"A_2760_MXZ02_O1"	Q 765.7	BOOL	// GERM FAN 2
"A_2801_MXZ01_O1"	Q 802.0	BOOL	// BELT CONVEYOR
"A_2802_MXZ01_O1"	Q 802.1	BOOL	// CHUTE DRIVE LEFT SIDE
"A_2802_MXZ01_O2"	Q 802.2	BOOL	// CHUTE DRIVE RIGHT SIDE
"A_2811_MXZ61_O1"	Q 803.2	BOOL	// TURNING SCREW DRIVE 1
"A_2811_MXZ62_O1"	Q 803.3	BOOL	// TURNING SCREW DRIVE 2
"A_2811_MXZ63_O1"	Q 803.4	BOOL	// TURNING SCREW DRIVE 3
"A_2811_MXZ64_O1"	Q 803.5	BOOL	// TURNING SCREW DRIVE 4
"A_2811_MXZ65_O1"	Q 803.6	BOOL	// TURNING SCREW DRIVE 5
"A_2811_MXZ66_O1"	Q 803.7	BOOL	// TURNING SCREW DRIVE 6
"A_2811_MXZ67_O1"	Q 804.0	BOOL	// TURNING SCREW DRIVE 7
"A_2811_MXZ68_O1"	Q 804.1	BOOL	// TURNING SCREW DRIVE 8
"A_2811_MXZ69_O1"	Q 804.2	BOOL	// TURNING SCREW DRIVE 9
"A_2811_MXZ70_O1"	Q 804.3	BOOL	// TURNING SCREW DRIVE 10
"A_2811_MXZ71_O1"	Q 804.4	BOOL	// TURNING SCREW DRIVE 11
"A_2811_MXZ72_O1"	Q 804.5	BOOL	// TURNING SCREW DRIVE 12
"A_2811_MXZ73_O1"	Q 804.6	BOOL	// TURNING SCREW DRIVE 13
"A_2815_MXZ11_O1"	Q 808.0	BOOL	// HORIZONTAL SCREW
"A_2815_MXZ15_O1"	Q 808.2	BOOL	// LIFTING SCREW
"A_2815_MXZ21_O1"	Q 808.3	BOOL	// LIFTING DEVICE DOWN
"A_2815_MXZ21_O2"	Q 808.4	BOOL	// LIFTING DEVICE UP
"A_2845_QXV21_O1"	Q 816.0	BOOL	// START COOLING UNIT GERMINATING
"A_2845_QXV31_O1"	Q 816.1	BOOL	// START COOLING UNIT GERMINATING
"A_2801_QXV21_O1"	Q 816.2	BOOL	// BALL VALVE SPRAY WATER OPEN
"A_2816_QXV12_O2"	Q 816.4	BOOL	// BALL VALVE SPRINKING WATER LINE
"A_2831_QXV12_O1"	Q 816.6	BOOL	// BALL VALVE AIR HUMIDIFICATION
"A_2831_QXV22_O1"	Q 816.7	BOOL	// BALL VALVE AIR HUMIDIFICATION
"A_2831_QXV12_O2"	Q 817.2	BOOL	// BALL VALVE VALVE HUMIDIFICATION
"A_2899_PAZ11_O1"	Q 818.0	BOOL	// ALARM HORN MACHINE
"A_2812_QXV12_O2"	Q 840.0	BOOL	// BALL VALVE SPRINKING WATER LINE 1
"A_28_A408Z1_O1"	Q 840.1	BOOL	// RESET ALARM
"A_2811_KCL01_O1"	Q 840.4	BOOL	// ALARM FLASHER
"A_2811_KCL01_O2"	Q 840.5	BOOL	// SPARE
"A_2811_MXZ21_O1"	Q 841.0	BOOL	// COUPLING DRIVE
"A_2811_MXZ21_O2"	Q 841.1	BOOL	// COUPLING DRIVE
"A_2811_MXZ25_O1"	Q 841.2	BOOL	// COUPLING DRIVE
"A_2811_MXZ25_O2"	Q 841.3	BOOL	// COUPLING DRIVE
"A_2811_MXZ31_O1"	Q 841.4	BOOL	// COUPLING DRIVE
"A_2811_MXZ31_O2"	Q 841.5	BOOL	// COUPLING DRIVE
"A_2811_MXZ35_O1"	Q 841.6	BOOL	// COUPLING DRIVE
"A_2811_MXZ35_O2"	Q 841.7	BOOL	// COUPLING DRIVE
"A_2815_KCL01_O1"	Q 860.0	BOOL	// BACKWALL LIFTED
"A_2815_KCL01_O2"	Q 860.1	BOOL	// BACKWALL LOWERED
"A_2815_KCL01_O3"	Q 860.2	BOOL	// UNCOUPLED
"A_2815_KCL01_O4"	Q 860.3	BOOL	// COUPLED
"A_2815_KCL01_O5"	Q 860.4	BOOL	// WALL LOCKED
"A_2815_KCL01_O6"	Q 860.5	BOOL	// WALL UNLOCKED
"A_2815_KCL01_O7"	Q 860.6	BOOL	// CLEANING FLAP 1/2
"A_2815_MXZ41_O1"	Q 861.0	BOOL	// COUPLING DRIVE
"A_2815_MXZ41_O2"	Q 861.1	BOOL	// COUPLING DRIVE
"A_2815_MXZ45_O1"	Q 861.2	BOOL	// COUPLING DRIVE
"A_2815_MXZ45_O2"	Q 861.3	BOOL	// COUPLING DRIVE
"A_2850_MXZ01_O1"	Q 864.0	BOOL	// AIR-FLAP 1 OPEN
"A_2850_MXZ01_O2"	Q 864.1	BOOL	// AIR-FLAP 1 CLOSE
"A_2851_MXZ01_O1"	Q 864.4	BOOL	// AIR-FLAP 2 OPEN
"A_2851_MXZ01_O2"	Q 864.5	BOOL	// AIR-FLAP 2 CLOSE
"A_2852_MXZ01_O1"	Q 865.0	BOOL	// AIR-FLAP 3 OPEN
"A_2852_MXZ01_O2"	Q 865.1	BOOL	// AIR-FLAP 3 CLOSE
"A_2854_MXZ01_O1"	Q 865.4	BOOL	// WATER PUMP 1
"A_2855_MXZ01_O1"	Q 865.5	BOOL	// WATER PUMP 2
"A_2860_MXZ01_O1"	Q 865.6	BOOL	// GERM FAN 1
"A_2860_MXZ02_O1"	Q 865.7	BOOL	// GERM FAN 2
"A_3111_MXZ11_O1"	Q 900.0	BOOL	// UN-/LOADING SCREW DISCHARGE
"A_3111_MXZ21_O1"	Q 900.1	BOOL	// LIFTING DRIVE 1 INSIDE LOWERING
"A_3111_MXZ21_O2"	Q 900.2	BOOL	// LIFTING DRIVE 1 INSIDE LIFTING
"A_3111_MXZ31_O1"	Q 900.3	BOOL	// LIFTING DRIVE 2 OUTSIDE LOWERING
"A_3111_MXZ31_O2"	Q 900.4	BOOL	// LIFTING DRIVE 2 OUTSIDE LIFTING
"A_3111_MXZ41_O1"	Q 900.5	BOOL	// TRAVELING DRIVE
"A_3115_MXZ11_O1"	Q 900.6	BOOL	// DISCHARGE FLAP CLOSE
"A_3115_MXZ11_O2"	Q 900.7	BOOL	// DISCHARGE FLAP OPEN
"A_3135_MXZ11_O1"	Q 901.0	BOOL	// LOUVER RECYCLE AIR 1 CLOSE
"A_3135_MXZ11_O2"	Q 901.1	BOOL	// LOUVER RECYCLE AIR 1 OPEN
"A_3136_MXZ11_O1"	Q 901.2	BOOL	// LOUVER RECYCLE AIR 2 CLOSE
"A_3136_MXZ11_O2"	Q 901.3	BOOL	// LOUVER RECYCLE AIR 2 OPEN
"A_3140_MXZ11_O1"	Q 901.4	BOOL	// LOUVER RECYCLE AIR 1 CLOSE
"A_3140_MXZ11_O2"	Q 901.5	BOOL	// LOUVER RECYCLE AIR 1 OPEN
"A_3141_MXZ11_O1"	Q 901.6	BOOL	// LOUVER RECYCLE AIR 2 CLOSE
"A_3141_MXZ11_O2"	Q 901.7	BOOL	// LOUVER RECYCLE AIR 2 OPEN
"A_3145_MXZ11_O1"	Q 902.0	BOOL	// LOUVER WITHERING AIR 1 CLOSE
"A_3145_MXZ11_O2"	Q 902.1	BOOL	// LOUVER WITHERING AIR 1 OPEN
"A_3146_MXZ11_O1"	Q 902.2	BOOL	// LOUVER WITHERING AIR 2 CLOSE
"A_3146_MXZ11_O2"	Q 902.3	BOOL	// LOUVER WITHERING AIR 2 OPEN
"A_3150_MXZ11_O1"	Q 902.4	BOOL	// LOUVER FRESH AIR 1 CLOSE
"A_3150_MXZ11_O2"	Q 902.5	BOOL	// LOUVER FRESH AIR 1 OPEN
"A_3151_MXZ11_O1"	Q 902.6	BOOL	// LOUVER FRESH AIR 2 CLOSE
"A_3151_MXZ11_O2"	Q 902.7	BOOL	// LOUVER FRESH AIR 2 OPEN
"A_3152_MXZ11_O1"	Q 903.0	BOOL	// LOUVER FRESH AIR 3 CLOSE
"A_3152_MXZ11_O2"	Q 903.1	BOOL	// LOUVER FRESH AIR 3 OPEN
"A_3153_MXZ11_O1"	Q 903.2	BOOL	// LOUVER FRESH AIR 4 CLOSE
"A_3153_MXZ11_O2"	Q 903.3	BOOL	// LOUVER FRESH AIR 4 OPEN
"A_3158_MXZ11_O1"	Q 903.4	BOOL	// LOUVER AIR HEATER 1 CLOSE
"A_3158_MXZ11_O2"	Q 903.5	BOOL	// LOUVER AIR HEATER 1 OPEN
"A_3159_MXZ11_O1"	Q 903.6	BOOL	// LOUVER AIR HEATER 2 CLOSE
"A_3159_MXZ11_O2"	Q 903.7	BOOL	// LOUVER AIR HEATER 2 OPEN
"A_3101_MXZ01_O1"	Q 904.0	BOOL	// OUTLET FLAP DRIVE CLOSE
"A_3101_MXZ01_O2"	Q 904.1	BOOL	// OUTLET FLAP DRIVE OPEN
"A_3161_KCL11_O1"	Q 916.0	BOOL	// BURNER 1 MAIN FAN RUNNING
"A_3161_KCL11_O2"	Q 916.1	BOOL	// BURNER 1 EXTERAL ON
"A_3161_KCL12_O1"	Q 917.0	BOOL	// BURNER 2 MAIN FAN RUNNING
"A_3161_KCL12_O2"	Q 917.1	BOOL	// BURNER 2 EXTERAL ON
"A_3199_PAZ11_O1"	Q 924.0	BOOL	// ALARM HORN
"A_3211_MXZ11_O1"	Q 1000.0	BOOL	// UN-/LOADING SCREW DISCHARGE
"A_3211_MXZ21_O1"	Q 1000.1	BOOL	// LIFTING DRIVE 1 INSIDE LOWERING
"A_3211_MXZ21_O2"	Q 1000.2	BOOL	// LIFTING DRIVE 1 INSIDE LIFTING
"A_3211_MXZ31_O1"	Q 1000.3	BOOL	// LIFTING DRIVE 2 OUTSIDE LOWERING
"A_3211_MXZ31_O2"	Q 1000.4	BOOL	// LIFTING DRIVE 2 OUTSIDE LIFTING
"A_3211_MXZ41_O1"	Q 1000.5	BOOL	// TRAVELING DRIVE
"A_3215_MXZ11_O1"	Q 1000.6	BOOL	// DISCHARGE FLAP CLOSE
"A_3215_MXZ11_O2"	Q 1000.7	BOOL	// DISCHARGE FLAP OPEN
"A_3235_MXZ11_O1"	Q 1001.0	BOOL	// LOUVER RECYCLE AIR 1 CLOSE
"A_3235_MXZ11_O2"	Q 1001.1	BOOL	// LOUVER RECYCLE AIR 1 OPEN
"A_3236_MXZ11_O1"	Q 1001.2	BOOL	// LOUVER RECYCLE AIR 2 CLOSE
"A_3236_MXZ11_O2"	Q 1001.3	BOOL	// LOUVER RECYCLE AIR 2 OPEN
"A_3240_MXZ11_O1"	Q 1001.4	BOOL	// LOUVER RECYCLE AIR 1 CLOSE
"A_3240_MXZ11_O2"	Q 1001.5	BOOL	// LOUVER RECYCLE AIR 1 OPEN
"A_3241_MXZ11_O1"	Q 1001.6	BOOL	// LOUVER RECYCLE AIR 2 CLOSE
"A_3241_MXZ11_O2"	Q 1001.7	BOOL	// LOUVER RECYCLE AIR 2 OPEN
"A_3245_MXZ11_O1"	Q 1002.0	BOOL	// LOUVER WITHERING AIR 1 CLOSE
"A_3245_MXZ11_O2"	Q 1002.1	BOOL	// LOUVER WITHERING AIR 1 OPEN
"A_3246_MXZ11_O1"	Q 1002.2	BOOL	// LOUVER WITHERING AIR 2 CLOSE
"A_3246_MXZ11_O2"	Q 1002.3	BOOL	// LOUVER WITHERING AIR 2 OPEN
"A_3250_MXZ11_O1"	Q 1002.4	BOOL	// LOUVER FRESH AIR 1 CLOSE
"A_3250_MXZ11_O2"	Q 1002.5	BOOL	// LOUVER FRESH AIR 1 OPEN
"A_3251_MXZ11_O1"	Q 1002.6	BOOL	// LOUVER FRESH AIR 2 CLOSE
"A_3251_MXZ11_O2"	Q 1002.7	BOOL	// LOUVER FRESH AIR 2 OPEN
"A_3252_MXZ11_O1"	Q 1003.0	BOOL	// LOUVER FRESH AIR 3 CLOSE
"A_3252_MXZ11_O2"	Q 1003.1	BOOL	// LOUVER FRESH AIR 3 OPEN
"A_3253_MXZ11_O1"	Q 1003.2	BOOL	// LOUVER FRESH AIR 4 CLOSE
"A_3253_MXZ11_O2"	Q 1003.3	BOOL	// LOUVER FRESH AIR 4 OPEN
"A_3258_MXZ11_O1"	Q 1003.4	BOOL	// LOUVER AIR HEATER 1 CLOSE
"A_3258_MXZ11_O2"	Q 1003.5	BOOL	// LOUVER AIR HEATER 1 OPEN
"A_3259_MXZ11_O1"	Q 1003.6	BOOL	// LOUVER AIR HEATER 2 CLOSE
"A_3259_MXZ11_O2"	Q 1003.7	BOOL	// LOUVER AIR HEATER 2 OPEN
"A_3201_MXZ01_O1"	Q 1004.0	BOOL	// OUTLET FLAP DRIVE CLOSE
"A_3201_MXZ01_O2"	Q 1004.1	BOOL	// OUTLET FLAP DRIVE OPEN
"A_3261_KCL11_O1"	Q 1016.0	BOOL	// BURNER 3 MAIN FAN RUNNING
"A_3261_KCL11_O2"	Q 1016.1	BOOL	// BURNER 3 EXTERAL ON
"A_3299_PAZ11_O1"	Q 1024.0	BOOL	// ALARM HORN
"A_1911_MXZ01_O1"	Q 1102.0	BOOL	// BELT CONVEYOR
"A_1915_MXZ01_O1"	Q 1102.1	BOOL	// BELT CONVEYOR
"A_1921_MXZ01_O1"	Q 1102.2	BOOL	// BELT CONVEYOR
"A_1931_MXZ01_O1"	Q 1102.3	BOOL	// BELT CONVEYOR
"A_1941_MXZ01_O1"	Q 1102.4	BOOL	// BELT CONVEYOR
"A_1942_MXZ01_O3"	Q 1102.5	BOOL	// CHUTE DRIVE LOW ROTARY SPEED
"A_1942_MXZ01_O1"	Q 1102.6	BOOL	// CHUTE DRIVE LEFT SIDE
"A_1942_MXZ01_O2"	Q 1102.7	BOOL	// CHUTE DRIVE RIGHT SIDE
"A_1999_PAZ11_O1"	Q 1104.0	BOOL	// ALARM HORN
"A_1911_QXV31_O1"	Q 1108.0	BOOL	// BALL VALVE SPRAY WATER OPEN
"A_1915_QXV31_O1"	Q 1108.1	BOOL	// BALL VALVE SPRAY WATER OPEN
"A_1921_QXV31_O1"	Q 1108.2	BOOL	// BALL VALVE SPRAY WATER OPEN
"A_2911_MXZ01_O1"	Q 1118.0	BOOL	// BELT CONVEYOR
"A_2914_MXZ01_O1"	Q 1118.1	BOOL	// BELT CONVEYOR
"A_2917_MXZ01_O1"	Q 1118.2	BOOL	// BELT CONVEYOR
"A_2920_MXZ01_O1"	Q 1118.3	BOOL	// BELT CONVEYOR
"A_2923_MXZ01_O1"	Q 1118.4	BOOL	// BELT CONVEYOR
"A_2926_MXZ01_O1"	Q 1118.5	BOOL	// BELT CONVEYOR
"A_2929_MXZ01_O1"	Q 1118.6	BOOL	// BELT CONVEYOR
"A_2932_MXZ01_02_O1"	Q 1119.1	BOOL	// BELT CONVEYOR DRIVE 1/2
"A_2935_MXZ01_O1"	Q 1119.2	BOOL	// BELT CONVEYOR RIGHT
"A_2935_MXZ01_O2"	Q 1119.3	BOOL	// BELT CONVEYOR LEFT
"A_2999_PAZ11_O1"	Q 1120.0	BOOL	// ALARM HORN
"A_2911_QXV31_O1"	Q 1124.0	BOOL	// BALL VALVE SPRAY WATER OPEN
"A_2914_QXV31_O1"	Q 1124.1	BOOL	// BALL VALVE SPRAY WATER OPEN
"A_2917_QXV31_O1"	Q 1124.2	BOOL	// BALL VALVE SPRAY WATER OPEN
"A_2920_QXV31_O1"	Q 1124.3	BOOL	// BALL VALVE SPRAY WATER OPEN
"A_2923_QXV31_O1"	Q 1124.4	BOOL	// BALL VALVE SPRAY WATER OPEN
"A_2935_QXV31_O1"	Q 1124.6	BOOL	// BALL VALVE SPRAY WATER OPEN
"A_2935_QXV41_O1"	Q 1124.7	BOOL	// BALL VALVE SPRAY WATER OPEN
"A_3911_MXZ01_O1"	Q 1134.0	BOOL	// CHAIN CONVEYOR
"A_3912_MXZ01_O1"	Q 1134.1	BOOL	// OUTLET FLAP DRIVE CLOSE
"A_3912_MXZ01_O2"	Q 1134.2	BOOL	// OUTLET FLAP DRIVE OPEN
"A_3914_MXZ01_O1"	Q 1134.3	BOOL	// FAN DRIVE "NOTUSED"
"A_3921_MXZ01_O1"	Q 1134.4	BOOL	// CHAIN CONVEYOR
"A_3922_MXZ01_O1"	Q 1134.5	BOOL	// OUTLET FLAP DRIVE CLOSE
"A_3922_MXZ01_O2"	Q 1134.6	BOOL	// OUTLET FLAP DRIVE OPEN
"A_3924_MXZ01_O1"	Q 1134.7	BOOL	// FAN DRIVE "NOTUSED"
"A_3930_MXZ01_O1"	Q 1135.0	BOOL	// ELEVATOR
"A_3932_MXZ01_O1"	Q 1135.1	BOOL	// FAN DRIVE "NOTUSED"
"A_3935_MXZ01_O1"	Q 1135.2	BOOL	// FLAP BOX DRIVE RIGHT SIDE
"A_3935_MXZ01_O2"	Q 1135.3	BOOL	// FLAP BOX DRIVE LEFT SIDE
"A_3938_MXZ01_O1"	Q 1135.4	BOOL	// BELT CONVEYOR
"A_3945_MXZ01_O1"	Q 1135.5	BOOL	// ELEVATOR
"A_3952_MXZ01_O1"	Q 1135.6	BOOL	// DISCHARGER DMBG DRIVE
"A_3955_MXZ01_O1"	Q 1135.7	BOOL	// SCREW CONVEYOR DRIVE
"A_3952_XCJ20_O1"	Q 1136.0	BOOL	// VALVE DMBG CLOSE
"A_3952_XCJ20_O2"	Q 1136.1	BOOL	// VALVE DMBG OPEN
"A_3952_XCJ20_O3"	Q 1136.2	BOOL	// VALVE DMBG CLOSE
"A_3952_XCJ20_O4"	Q 1136.3	BOOL	// VALVE DMBG OPEN
"A_3960_MXZ01_O1"	Q 1136.4	BOOL	// FAN DRIVE
"A_3965_MXZ01_O1"	Q 1136.5	BOOL	// AIRLOCK
"A_3970_MXZ01_O1"	Q 1136.6	BOOL	// AIRLOCK
"A_3999_PAZ11_O1"	Q 1137.0	BOOL	// ALARM HORN
"A_3913_KFC10_O1"	Q 1140.0	BOOL	// FILTER ASPIRATION ON "NOTUSED"
"A_3923_KFC10_O1"	Q 1140.1	BOOL	// FILTER ASPIRATION ON "NOTUSED"
"A_3931_KFC10_O1"	Q 1140.2	BOOL	// FILTER ASPIRATION ON "NOTUSED"
"A_3956_KCL01_O2"	Q 1140.4	BOOL	// LIGHT CUSTOMER ON
"A_3956_KCL01_O3"	Q 1140.5	BOOL	// LIGHT CUSTOMER OFF
"A_3956_KCL01_O1"	Q 1140.6	BOOL	// TURN ON EXCISTING DEGERMINATING SYSTEM
"A_2145_QXV21_AO1"	QW 168	WORD	// REGULATING VALVE SET POINT
"A_2145_QXV31_AO1"	QW 170	WORD	// REGULATING VALVE SET POINT
"A_2245_QXV21_AO1"	QW 268	WORD	// REGULATING VALVE SET POINT
"A_2245_QXV31_AO1"	QW 270	WORD	// REGULATING VALVE SET POINT
"A_2345_QXV21_AO1"	QW 368	WORD	// REGULATING VALVE SET POINT
"A_2345_QXV31_AO1"	QW 382	WORD	// REGULATING VALVE SET POINT
"A_2445_QXV21_AO1"	QW 468	WORD	// REGULATING VALVE SET POINT
"A_2445_QXV31_AO1"	QW 482	WORD	// REGULATING VALVE SET POINT
"CTUD"	SFB 2	SFB 2	// Count Up / Down
"TON"	SFB 4	SFB 4	// Generate an On Delay
"SIEMENS_BSEND"	SFB 12	SFB 12	// SIEMENS: Block Oriented Send
"SIEMENS_BRCV"	SFB 13	SFB 13	// SIEMENS: Block Oriented Receive
"SIEMENS_HS_COUNT"	SFB 29	SFB 29	// SIEMENS: High-Speed Counter (CPU 312, Integrated Function)
"SIEMENS_FREQ_MES"	SFB 30	SFB 30	// SIEMENS: Frequency Meter (CPU 312, Integrated Function)
"SIEMENS_POSITION"	SFB 31	SFB 31	// SIEMENS: Open-Loop Positioning (CPU 312, Integrated Function)
"SIEMENS_SET_CLK"	SFC 0	SFC 0	// SIEMENS: Set System Clock
"SIEMENS_READ_CLK"	SFC 1	SFC 1	// SIEMENS: Read System Clock
"SIEMENS_SET_RTM"	SFC 2	SFC 2	// SIEMENS: Set Run-Time Meter
"SIEMENS_CTRL_RTM"	SFC 3	SFC 3	// SIEMENS: Start/Stop Run-Time Meter
"SIEMENS_READ_RTM"	SFC 4	SFC 4	// SIEMENS: Read Run-Time Meter
"GADR_LGC"	SFC 5	SFC 5	// Query Logical Address of a Channel
"RD_SINFO"	SFC 6	SFC 6	// Read OB Start Information
"DPNRM_DG"	SFC 13	SFC 13	// Read Diagnostic Data of a DP Slave
"SIEMENS_DPRD_DAT"	SFC 14	SFC 14	// SIEMENS: Read data for DP-Node
"SIEMENS_DPWR_DAT"	SFC 15	SFC 15	// SIEMENS: Write Data to DP-Node
"SIEMENS_BLKMOV"	SFC 20	SFC 20	// SIEMENS: Direct Word Move
"SIEMENS_FILL"	SFC 21	SFC 21	// SIEMENS: Initialize a memory area
"SIEMENS_CREAT_DB"	SFC 22	SFC 22	// SIEMENS: Create Data Block
"SIEMENS_TEST_DB"	SFC 24	SFC 24	// SIEMENS: Test DB
"SIEMENS_SET_TINT"	SFC 28	SFC 28	// SIEMENS: Set Time-of-Day Interrupt
"SIEMENS_CAN_TINT"	SFC 29	SFC 29	// SIEMENS: Cancel Time-of-Day Interrupt
"SIEMENS_ACT_TINT"	SFC 30	SFC 30	// SIEMENS: Activate Time-of-Day Interrupt
"SIEMENS_QRY_TINT"	SFC 31	SFC 31	// SIEMENS: Query Time-of-Day Interrupt
"SIEMENS_SRT_DINT"	SFC 32	SFC 32	// SIEMENS: Start Time-Delay Interrupt
"SIEMENS_CAN_DINT"	SFC 33	SFC 33	// SIEMENS: Cancel Time-Delay Interrupt
"SIEMENS_QRY_DINT"	SFC 34	SFC 34	// SIEMENS: Query Time-Delay Interrupt
"SIEMENS_MSK_FLT"	SFC 36	SFC 36	// SIEMENS: Mask synchronous faults
"SIEMENS_DMSK_FLT"	SFC 37	SFC 37	// SIEMENS: Unmask Synchronous Faults
"SIEMENS_READ_ERR"	SFC 38	SFC 38	// SIEMENS: Read Error Registers
"SIEMENS_DIS_IRT"	SFC 39	SFC 39	// SIEMENS: Disable Interrupt
"SIEMENS_EN_IRT"	SFC 40	SFC 40	// SIEMENS: Enable New Interrupts and Asynchronous Errors
"SIEMENS_DIS_AIRT"	SFC 41	SFC 41	// SIEMENS: Disable Alarm Interrupts
"SIEMENS_EN_AIRT"	SFC 42	SFC 42	// SIEMENS: Enable Alarm Interrupts
"SIEMENS_RE_TRIGR"	SFC 43	SFC 43	// SIEMENS: Retrigger Cycle Time Monitoring
"SIEMENS_REPL_VAL"	SFC 44	SFC 44	// SIEMENS: Replace Value
"SIEMENS_STP"	SFC 46	SFC 46	// SIEMENS: Change the CPU to STOP
"SIEMENS_WAIT"	SFC 47	SFC 47	// SIEMENS: Wait
"SIEMENS_LGC_GADR"	SFC 49	SFC 49	// SIEMENS:
"SIEMENS_RD_LGADR"	SFC 50	SFC 50	// SIEMENS:
"SIEMENS_RDSYSST"	SFC 51	SFC 51	// SIEMENS: Read System Status
"SIEMENS_WR_USMSG"	SFC 52	SFC 52	// SIEMENS: Write User Element in Diagnosis Buffer
"SIEMENS_WR_PARM"	SFC 55	SFC 55	// SIEMENS: Synchronous Write Parameter (MC7)
"SIEMENS_WR_DPARM"	SFC 56	SFC 56	// SIEMENS: Synchronous Write Parameter (SDB)
"SIEMENS_PARM_MOD"	SFC 57	SFC 57	// SIEMENS: Synchronous Write Static and Dynamic
"SIEMENS_WR_REC"	SFC 58	SFC 58	// SIEMENS: Write Data Record
"SIEMENS_RD_REC"	SFC 59	SFC 59	// SIEMENS: Read Data Record
"SIEMENS_AB_CALL"	SFC 63	SFC 63	// SIEMENS: Assembly Code Block (CPU 614)
"SIEMENS_TIME_TCK"	SFC 64	SFC 64	// SIEMENS: Time Tick
"SYS_PLCStartUpDelay"	T 10	TIMER	// SYS: Delay software enable after plc startup
"SYS_HWDelay"	T 11	TIMER	// SYS: Delay software enable after hardware stop
"SYS_T_LOGEntryDelay"	T 13	TIMER	// SYS: Delay log entrys after fuse tripped
"SYS_T_OfflineDelay"	T 14	TIMER	// SYS: Delay section staOffline
"SYS_T_NStartOfflineTime"	T 15	TIMER	// SYS: Offline time after a newstart
"SYS_DelayHeavyStartup"	T 16	TIMER	// SYS: Monitoring time to reset flag
"SYS_DelayBrakeMill"	T 17	TIMER	// SYS: Monitoring time to reset flag brake mill
"COM_T_PCCWatchdog"	T 20	TIMER	// COM: Communication monitoring to process control computer
"SEW_MOVIDRIVE"	UDT 200	UDT 200	// MOVIDRIVE DFP21 (DPV1)
"DANFOSS_VLT5000"	UDT 203	UDT 203	// Danfoss VLT 5000
"ABB_ACS800"	UDT 204	UDT 204	// ABB ACS800 / RPBA-01
"NORDAC"	UDT 205	UDT 205	// NORDAC_SK500_SK TU3-PBR
"ASW_Flags_F0_F15"	UDT 1000	UDT 1000
"ASW_LineAnimation"	UDT 1001	UDT 1001
"ASW_UserSectionState"	UDT 1002	UDT 1002
"ASW_ProductInfo"	UDT 1003	UDT 1003
"SSA_HandAddInfo"	UDT 1004	UDT 1004
"ASW_DFCARecipe"	UDT 1005	UDT 1005
"SSA_MH_ProcessTime"	UDT 2000	UDT 2000	// Malthouse Actual time Process
"SSA_MH_StepTime"	UDT 2001	UDT 2001	// Malthouse Actual time Step
"SSA_MH_JobHeader"	UDT 2003	UDT 2003	// Malthouse SecNom: Job_Header
"SSA_MH_SecNomStandPIC"	UDT 2004	UDT 2004	// Malthouse SecNom: Standard Command PC
"SSA_MH_Step_Loading"	UDT 2011	UDT 2011	// Malthouse Step Loading
"SSA_MH_Step_Unloading"	UDT 2012	UDT 2012	// Malthouse Step Unloading
"SSA_MH_Step_Clearing"	UDT 2013	UDT 2013	// Malthouse Step Clearing
"SSA_Steep_Cmd"	UDT 2100	UDT 2100	// Steeping Section: Commands
"SSA_Steep_Par"	UDT 2101	UDT 2101	// Steeping Section: Parameter
"SSA_Steep_Recipe"	UDT 2102	UDT 2102	// Steeping Section: Recipe
"SSA_Steep_Analog"	UDT 2103	UDT 2103	// Steeping Section: Analog Values
"SSA_Steep_Recipe_Header"	UDT 2104	UDT 2104	// Steeping Section: Recipe Header
"SSA_Steep_Step"	UDT 2105	UDT 2105	// Steeping Section : Single Step
"SSA_Steep_Sum"	UDT 2106	UDT 2106	// Summary values for Steeping with sequencial conical steep
"SSA_Germ_Cmd"	UDT 2200	UDT 2200	// Germination Section: Commands
"SSA_Germ_Par"	UDT 2201	UDT 2201	// Germination Section: Parameter
"SSA_Germ_Recipe"	UDT 2202	UDT 2202	// Germination Section: Recipe
"SSA_Germ_Analog"	UDT 2203	UDT 2203	// Germination Section: Analog Values
"SSA_Germ_Recipe_Header"	UDT 2204	UDT 2204	// Germination Section:  Recipe Header
"SSA_Germ_Step"	UDT 2205	UDT 2205	// Germination Section: Single Step
"SSA_Kiln_Cmd"	UDT 2300	UDT 2300	// Kilning Section: Commands
"SSA_Kiln_Par"	UDT 2301	UDT 2301	// Kilning Section: Parameter
"SSA_Kiln_Recipe"	UDT 2302	UDT 2302	// Kilning Section: Recipe
"SSA_Kiln_Analog"	UDT 2303	UDT 2303	// Kilning Section: Analog Values
"SSA_Kiln_Recipe_Header"	UDT 2304	UDT 2304	// Kilning Section:  Recipe Header
"SSA_Kiln_Step"	UDT 2305	UDT 2305	// Kilning Section: Single Step
"UDTL01LineCmd"	UDT 3200	UDT 3200
"UDTL01SecData"	UDT 3202	UDT 3202
"UDTL01SecAc"	UDT 3203	UDT 3203
"UDTL01SecNom"	UDT 3204	UDT 3204
"ASW_MAL1OnOffCmd"	UDT 8000	UDT 8000	// ASW: Line Command
"ASW_MAL1SecNom"	UDT 8001	UDT 8001	// ASW: Nominal Data
"ASW_MAL1SecAc"	UDT 8002	UDT 8002	// ASW: Actual Data
"CMDs_ILO_Funktion"	UDT 8015	UDT 8015	// Command and setpoints for one ILO-funktion
"SSA_LOG_Value"	UDT 10005	UDT 10005
"ASW_CBitDeclaration"	UDT 10020	UDT 10020	// ASW: Declaration of change bit data blocks
"GCS7_UDT_Timer"	UDT 10180	UDT 10180	// Timer in DB
"CWA_UDT_Command"	UDT 10413	UDT 10413	// UDT Command  for CWA
"CWA_UDT_BinParaShort"	UDT 10418	UDT 10418	// UDT CWA bin parameter with minimum used parameter
"CWA_UDT_BinParaAll"	UDT 10419	UDT 10419	// UDT CWA bin parameter with all parameters
"GCS7_UDT_FunctionKey"	UDT 10601	UDT 10601	// GCS7: Upper Layer
"GCS7_UDT_FaultPattern"	UDT 10602	UDT 10602	// GCS7: Upper Layer
"GCS7_UDT_StatusPattern"	UDT 10603	UDT 10603	// Upper Layer
"GCS7_UDT_BINList1"	UDT 10660	UDT 10660	// GCS7: Binlist without WtActual and WtTarget
"GCS7_UDT_BINStatus"	UDT 10662	UDT 10662	// GCS7: Binstatus
"GCS7_UDT_BINList2"	UDT 10664	UDT 10664	// GCS7: Binlist with WtActual without WtTarget
"GCS7_UDT_BINList3"	UDT 10668	UDT 10668	// GCS7: Binlist with WtActual and WtTarget
"GCS7_UDT_ScaleControl"	UDT 10680	UDT 10680	// GCS7: Scale control
"ASW_StageCtrl"	UDT 18000	UDT 18000
"PCCYieldScale"	UDT 19000	UDT 19000	// USW: Struct for scales involved in yield calculation
"WinCoSYieldScale"	UDT 19001	UDT 19001	// USW: Struct for scales involved in yield calculation
"SamplerData"	UDT 19002	UDT 19002	// USW: Struct for sampler data
"BigBagData"	UDT 19003	UDT 19003	// Registration of big bag weight
"GCS7_FB9_Section"	UDT 20090	UDT 20090	// Group Control: Interface Section
"GCS7_GR_COM"	UDT 20097	UDT 20097	// GCS7 Data PLC Communication per group
"GCS90S7_FB9_Communicat"	UDT 20098	UDT 20098	// Communication PLC --PLC GCS7 to GCS90S7
"GCS7_FB9_Communication"	UDT 20099	UDT 20099	// Communication PLC --PLC
"GCS7_FB11_Communication"	UDT 20119	UDT 20119	// Communication PLC --PLC
"GCS7_FB12_Communication"	UDT 20129	UDT 20129	// Communication PLC --PLC
"GCS7_FB13_Communication"	UDT 20139	UDT 20139	// Communication PLC --PLC
"GCS7_FB14_Communication"	UDT 20149	UDT 20149	// Communication PLC --PLC
"GCS7_FB16_Communication"	UDT 20169	UDT 20169	// Communication PLC --PLC
"GCS7_FB37_DP_Alarm"	UDT 20373	UDT 20373	// SSW: Element MDDR/T Alarms
"GCS7_FB40_dynData"	UDT 20400	UDT 20400	// Lower Layer
"GCS7_M_FB41_Data"	UDT 20410	UDT 20410	// Lower Layer
"GCS7_M_FB44_Data"	UDT 20440	UDT 20440	// Lower Layer
"GCS7_M_FB45_Data"	UDT 20450	UDT 20450	// Lower Layer
"GCS7_M_FB46_Data"	UDT 20460	UDT 20460	// Lower Layer
"GCS7_M_FB47_Data"	UDT 20470	UDT 20470	// Lower Layer
"GCS7_M_FB48_Data"	UDT 20480	UDT 20480	// Lower Layer
"GCS7_M_FB49_Data"	UDT 20490	UDT 20490	// Lower Layer
"GCS7_M_FB50_Data"	UDT 20500	UDT 20500	// Lower Layer
"GCS7_M_FB51_Data"	UDT 20510	UDT 20510	// Lower Layer
"GCS7_M_FB52_Data"	UDT 20520	UDT 20520	// Lower Layer
"GCS7_M_FB53_Data"	UDT 20530	UDT 20530	// Lower Layer
"GCS7_M_FB54_Data"	UDT 20540	UDT 20540	// Lower Layer
"GCS7_M_FB55_Data"	UDT 20550	UDT 20550	// Lower Layer
"GCS7_M_FB56_Data"	UDT 20560	UDT 20560	// Lower Layer
"GCS7_M_FB58_Data"	UDT 20580	UDT 20580	// Lower Layer
"GCS7_M_FB59_Data"	UDT 20590	UDT 20590	// Lower Layer
"GCS7_M_FB60_Data"	UDT 20600	UDT 20600	// Lower Layer
"GCS7_M_FB61_Data"	UDT 20610	UDT 20610	// Lower Layer
"GCS7_M_FB62_Data"	UDT 20620	UDT 20620	// Lower Layer
"GCS7_M_FB63_Data"	UDT 20630	UDT 20630	// Lower Layer
"GCS7_M_FB64_Data"	UDT 20640	UDT 20640	// Lower Layer
"GCS7_M_FB65_Data"	UDT 20650	UDT 20650	// Lower Layer
"GCS7_M_FB66_Data"	UDT 20660	UDT 20660	// Lower Layer
"GCS7_M_FB67_Data"	UDT 20670	UDT 20670	// Lower Layer
"GCS7_M_FB68_Data"	UDT 20680	UDT 20680	// Lower Layer
"GCS7_M_FB69_Data"	UDT 20690	UDT 20690	// Lower Layer
"GCS7_E_FB73_A201"	UDT 20735	UDT 20735	// DFCA: Data Telegram A201:
"GCS7_M_FB81_Data"	UDT 20810	UDT 20810	// Lower Layer
"GCS7_M_FB82_Data"	UDT 20820	UDT 20820	// Lower Layer
"GCS7_FB84_Communication"	UDT 20849	UDT 20849	// Communication PLC --PLC
"GCS7_FB85_Data"	UDT 20850	UDT 20850	// Stroke Drive
"GCS7_FB85_Counter"	UDT 20851	UDT 20851	// Data of Increment counter
"GCS7_FB86_Data"	UDT 20860	UDT 20860
"GCS7_M_FB87_Data"	UDT 20870	UDT 20870	// Machine 4/8 roll stand with profibus
"GCS7_M_FB88_Data"	UDT 20880	UDT 20880	// Machin Flat-bottom discharger
"GR052_UDT"	UDT 21520	UDT 21520	// UDT way groupAspiration Flaps Bin 21 to 34 (Aspiration)
"SSW_EL_ASI_Slave"	UDT 28995	UDT 28995	// Element Control ASI Master Wago/Profibus Slave Data
"ASW_UDTOnOffCmd"	UDT 32700	UDT 32700
"ASW_UDTSecNom"	UDT 32701	UDT 32701	// Nominal value for section
"ASW_UDTSecAc"	UDT 32702	UDT 32702	// Actual values of section
END_SYMBOL_TABLE
